{attribute 'qualified_only'}
VAR_GLOBAL
	IBN_bool: ARRAY[1..16] OF BOOL;
	IBN_int: ARRAY[1..16] OF INT;
	IBN_dint: ARRAY[1..16] OF DINT;
	IBN_udint: ARRAY[1..16] OF UDINT;
	IBN_Timer: ARRAY[1..16] OF TON; 
END_VAR

(* stored: Version 1.1.0.1
   GVL Debug: Id {edbc2757-db55-4a3c-881b-283dd95aa9d9} *)
